        print(f"Attempting to join: {face_target_name} to {pickup_target_name} as {program_name_to_pickup}")
        # Call the plugin command to join the face target to the pickup target
        status_to_pickup = RDK.PluginCommand(
            "CollisionFreePlanner",
            "Join",
            f"{face_target_name}|{pickup_target_name}|{program_name_to_pickup}"
        )
        print(f"Status for '{program_name_to_pickup}': {status_to_pickup}")

        # --- Check and delete existing "From Pickup" program ---
        existing_prog_from_pickup = RDK.Item(program_name_from_pickup, ITEM_TYPE_PROGRAM)
        if existing_prog_from_pickup.Valid():
            print(f"Deleting existing program: {program_name_from_pickup}")
            existing_prog_from_pickup.Delete()

        print(f"Attempting to join: {pickup_target_name} to {face_target_name} as {program_name_from_pickup}")
        # Call the plugin command to join the pickup target to the face target
        status_from_pickup = RDK.PluginCommand(
            "CollisionFreePlanner",
            "Join",
            f"{pickup_target_name}|{face_target_name}|{program_name_from_pickup}"
        )
        print(f"Status for '{program_name_from_pickup}': {status_from_pickup}")


    print("\nPickup link generation process finished.")


# --- Main execution: Run only the new functions ---
if __name__ == '__main__':
    create_face_targets()
    generate_pickup_links()
    create_face_programs()
    addmainprogram()

--- Python program ProgramGenerator ---
from robodk import robolink

# Connect to RoboDK
RDK = robolink.Robolink()

# Get the robot, reference frame, and base point
robot = RDK.Item('UR10e')  # Replace 'Robot' with your robot's name
reference_frame = RDK.Item('CSV Frame')  # Replace 'Reference Frame' with your frame's name
base_point = RDK.Item('Target 33')  # Replace 'Point 1' with your base point's name

# Create a new program
program = RDK.AddProgram('AutoProgram')

# Get all targets under the reference frame
targets = reference_frame.Childs()
target_list = [target for target in targets if target.Type() == robolink.ITEM_TYPE_TARGET]

# Add movements and screwdriver actions to the program
for i, target in enumerate(target_list):
    # Move to the base point first (except for the first target)
    if i > 0:
        program.MoveL(base_point)

    # Move to the target point
    program.MoveL(target)

    # Execute screwdriver actions
    program.RunInstruction('move_shank(20)', robolink.INSTRUCTION_CALL_PROGRAM)  # Tighten screw
    program.RunInstruction('move_shank(0)', robolink.INSTRUCTION_CALL_PROGRAM)  # Release screwdriver

# Save the program
#program.ShowTargets(False)  # Hide targets for clarity
program.Update()
print("Program generated successfully!")

--- Python program ProgramGenerator ---
from robodk import robolink

# Connect to RoboDK
RDK = robolink.Robolink()

# Get the robot, reference frame, and base point
robot = RDK.Item('UR10e')  # Replace 'Robot' with your robot's name
reference_frame = RDK.Item('CSV Frame')  # Replace 'Reference Frame' with your frame's name
base_point = RDK.Item('Target 33')  # Replace 'Point 1' with your base point's name

# Create a new program
program = RDK.AddProgram('AutoProgram')

# Get all targets under the reference frame
targets = reference_frame.Childs()
target_list = [target for target in targets if target.Type() == robolink.ITEM_TYPE_TARGET]

# Add movements and screwdriver actions to the program
for i, target in enumerate(target_list):
    # Move to the base point first (except for the first target)
    if i > 0:
        program.MoveL(base_point)

    # Move to the target point
    program.MoveL(target)

    # Execute screwdriver actions
    program.RunInstruction('move_shank(20)', robolink.INSTRUCTION_CALL_PROGRAM)  # Tighten screw
    program.RunInstruction('move_shank(0)', robolink.INSTRUCTION_CALL_PROGRAM)  # Release screwdriver

# Save the program
#program.ShowTargets(False)  # Hide targets for clarity
program.Update()
print("Program generated successfully!")

--- program pickupm5Totoolswitchm8approach (robot UR10e) ---
  MoveJ (Pt 1 (S1138)) to (-437.91, 304.62, 83.06) mm, rotated rx 148.82 ry 3.26 rz -178.93 deg; joints [-75.565, -105.059, 145.828, -26.927, 13.754, -134.641]
  MoveJ (Pt 2 (S1069)) to (-424.05, 221.6, 32.68) mm, rotated rx 148.94 ry 3.77 rz -174.12 deg; joints [-76.807, -103.326, 153.048, -22.371, 8.218, -148.169]
  MoveJ (Pt 3 (S995)) to (-436.51, 254.57, 169.63) mm, rotated rx 148.94 ry 3.77 rz -174.12 deg; joints [-75.55, -113.946, 140.961, -3.178, 9.351, -144.613]
  MoveJ (Pt 4 (S1013)) to (-349.4, 349.66, 227.68) mm, rotated rx 175.61 ry -30.98 rz 98.15 deg; joints [-40.94, -114.594, 151.115, -74.991, 124.156, -118.436]
  MoveJ (Pt 5 (S876)) to (-566.01, -9.66, 385.13) mm, rotated rx 90 ry -10 rz -90 deg; joints [-56.219, -97.868, 132.397, -22.553, -56.798, -186.625]
  MoveJ (Pt 6 (S768)) to (-566.01, -53.07, 388.93) mm, rotated rx 90 ry 0 rz -90 deg; joints [-52.421, -105.764, 133.113, -27.35, -52.42, -179.999]
  MoveJ (Pt 7 (S516)) to (-566.01, -172.58, 395.39) mm, rotated rx 90 ry 0 rz -90 deg; joints [-37.286, -110.687, 135.476, -24.792, -37.284, -179.998]
  MoveJ (Pt 8 (S386)) to (-566.01, -242.72, 394.37) mm, rotated rx 90 ry 0 rz -90 deg; joints [-25.901, -110.898, 135.712, -24.817, -25.9, -179.997]
  MoveJ (Pt 9 (S229)) to (-566.01, -361.29, 394.37) mm, rotated rx 90 ry 0 rz -90 deg; joints [-5.068, -107.128, 133.402, -26.287, -5.067, -179.986]
  MoveJ (Pt 10 (S154)) to (-816.01, -361.29, 394.37) mm, rotated rx 90 ry 0 rz -90 deg; joints [-2.904, -81.882, 110.532, -28.675, -2.903, -179.976]
  MoveJ (Pt 11 (S109)) to (-816.02, -422.58, 395.39) mm, rotated rx 90 ry 0 rz -90 deg; joints [2.982, -80.355, 108.601, -28.223, 2.983, -180.023]
  MoveJ (Pt 12 (S93)) to (-624.17, -467.56, 176.05) mm, rotated rx -179.87 ry 0.01 rz -89.96 deg; joints [6.858, -76.682, 103.853, 332.885, 6.813, -89.924]
  MoveJ (Pt 13 (S142)) to (-623.94, -467.54, 76.05) mm, rotated rx -179.87 ry 0.01 rz -89.96 deg; joints [6.859, -71.505, 108.744, 322.817, 6.815, -89.924]

--- program Program_Main_Combined_met (robot UR10e) ---
  Set Tool: schroevendraaier all in met nieuw kopstuk en tool
  Set Ref.: CSV Frame
  Call pickupm8Totoolswitchm8approach
  Call toolswitchm8approachTopickupm8
  Call Program_Main_m8
  Call pickupm8Totoolswitchm8approach
  Call toolswitchm8approachTopickupm8

--- program Program_Main_Combined_met (robot UR10e) ---
  Set Tool: schroevendraaier all in met nieuw kopstuk en tool
  Set Ref.: CSV Frame
  Call pickupm8Totoolswitchm8approach
  MoveL (toolswitch_m8)
  Call screw_out(0)
  MoveL (toolswitch_m8_approach)
  Call toolswitchm8approachTopickupm8
  Call Program_Main_m8
  Call pickupm8Totoolswitchm8approach
  MoveL (toolswitch_m8)
  Call screw_in(10)
  MoveL (toolswitch_m8_approach)
  Call toolswitchm8approachTopickupm8

--- program Program_Main_Combined_met (robot UR10e) ---
  Set Tool: schroevendraaier all in met nieuw kopstuk en tool
  Set Ref.: CSV Frame

--- program Prog43 (robot UR10e) ---
  Set Ref.: CSV Frame
  Set Tool: schroevendraaier all in met nieuw kopstuk en tool
  MoveL (toolswitch_m8_approach)
  MoveL (toolswitch_m8)
  Call screw_out(0)
  MoveL (toolswitch_m8_approach)
  MoveL (toolswitch_m8_approach)
  MoveL (toolswitch_m8)
  Call screw_in(10)
  MoveL (toolswitch_m8_approach)

--- program pickupm8Totoolswitchm8 (robot UR10e) ---
  MoveJ (Pt 1 (S1265)) to (-361.97, 306.04, 87.38) mm, rotated rx 148.82 ry 3.26 rz -178.93 deg; joints [-96.274, -127.938, 155.828, 308.074, -8.028, -97.355]
  MoveJ (Pt 2 (S1276)) to (-291.81, 189.68, 43.36) mm, rotated rx 173.25 ry 30.68 rz -107.38 deg; joints [-75.824, -114.001, 145.678, 293.478, -63.249, -79.354]
  MoveJ (Pt 3 (S1105)) to (-362.69, 295.7, 104.49) mm, rotated rx 173.25 ry 30.68 rz -107.38 deg; joints [-70.201, -101.671, 131.181, 293.82, -58.685, -75.597]
  MoveJ (Pt 4 (S1048)) to (-433.56, 401.71, 165.63) mm, rotated rx 173.25 ry 30.68 rz -107.38 deg; joints [-67.129, -91.484, 115.69, 297.937, -56.239, -73.391]
  MoveJ (Pt 5 (S1116)) to (-437.47, 349.85, 251.04) mm, rotated rx 173.25 ry 30.68 rz -107.38 deg; joints [-64.592, -98.205, 112.824, 306.43, -54.251, -71.473]
  MoveJ (Pt 6 (S1022)) to (-463.16, 267.77, 200.01) mm, rotated rx 173.25 ry 30.68 rz -107.38 deg; joints [-57.766, -100.913, 120.893, 297.542, -49.071, -65.796]
  MoveJ (Pt 7 (S999)) to (-488.86, 185.69, 148.99) mm, rotated rx 173.25 ry 30.68 rz -107.38 deg; joints [-49.635, -101.874, 128.097, 285.751, -43.336, -57.797]
  MoveJ (Pt 8 (S918)) to (-484.94, 237.56, 63.59) mm, rotated rx 173.25 ry 30.68 rz -107.38 deg; joints [-53.767, -93.623, 130.789, 277.833, -46.181, -62.054]
  MoveJ (Pt 9 (S905)) to (-484.22, 247.88, 46.49) mm, rotated rx 173.24 ry 30.67 rz -107.38 deg; joints [-54.525, -91.744, 131.117, 276.144, -46.717, -62.802]
  MoveJ (Pt 10 (S31)) to (-569.54, 226.04, 79.52) mm, rotated rx -176.96 ry 3.26 rz -178.93 deg; joints [-56.803, -92.592, 131.94, -33.233, 32.278, -92.138]
  MoveJ (Pt 11 (S27)) to (-580.12, 225.84, 78.92) mm, rotated rx -176.96 ry 3.26 rz -178.93 deg; joints [-55.548, -91.667, 131.136, -33.557, 33.527, -91.896]
  MoveJ (Pt 12 (S28)) to (-581.67, 325.69, 73.63) mm, rotated rx -176.96 ry 3.26 rz -178.93 deg; joints [-62.052, -84.921, 124.838, -32.736, 27.065, -93.365]

--- program toolswitchm8Topickupm8 (robot UR10e) ---
  MoveJ (Pt 1 (S28)) to (-581.67, 325.69, 73.63) mm, rotated rx -176.96 ry 3.26 rz -178.93 deg; joints [-62.052, -84.921, 124.838, -32.736, 27.065, -93.365]
  MoveJ (Pt 2 (S27)) to (-580.12, 225.84, 78.92) mm, rotated rx -176.96 ry 3.26 rz -178.93 deg; joints [-55.548, -91.667, 131.136, -33.557, 33.527, -91.896]
  MoveJ (Pt 3 (S31)) to (-569.54, 226.04, 79.52) mm, rotated rx -176.96 ry 3.26 rz -178.93 deg; joints [-56.803, -92.592, 131.94, -33.233, 32.278, -92.138]
  MoveJ (Pt 4 (S905)) to (-484.22, 247.88, 46.49) mm, rotated rx 173.24 ry 30.67 rz -107.38 deg; joints [-54.525, -91.744, 131.117, 276.144, -46.717, -62.802]
  MoveJ (Pt 5 (S975)) to (-488.13, 196.03, 131.91) mm, rotated rx 173.24 ry 30.67 rz -107.38 deg; joints [-50.502, -100.38, 128.761, 284.277, -43.917, -58.739]
  MoveJ (Pt 6 (S999)) to (-488.86, 185.69, 148.99) mm, rotated rx 173.25 ry 30.68 rz -107.38 deg; joints [-49.635, -101.874, 128.097, 285.751, -43.336, -57.797]
  MoveJ (Pt 7 (S1022)) to (-463.16, 267.77, 200.01) mm, rotated rx 173.25 ry 30.68 rz -107.38 deg; joints [-57.766, -100.913, 120.893, 297.542, -49.071, -65.796]
  MoveJ (Pt 8 (S1116)) to (-437.47, 349.85, 251.04) mm, rotated rx 173.25 ry 30.68 rz -107.38 deg; joints [-64.592, -98.205, 112.824, 306.43, -54.251, -71.473]
  MoveJ (Pt 9 (S1048)) to (-433.56, 401.71, 165.63) mm, rotated rx 173.25 ry 30.68 rz -107.38 deg; joints [-67.129, -91.484, 115.69, 297.937, -56.239, -73.391]
  MoveJ (Pt 10 (S1105)) to (-362.69, 295.7, 104.49) mm, rotated rx 173.25 ry 30.68 rz -107.38 deg; joints [-70.201, -101.671, 131.181, 293.82, -58.685, -75.597]
  MoveJ (Pt 11 (S1276)) to (-291.81, 189.68, 43.36) mm, rotated rx 173.25 ry 30.68 rz -107.38 deg; joints [-75.824, -114.001, 145.678, 293.478, -63.249, -79.354]
  MoveJ (Pt 12 (S1265)) to (-361.97, 306.04, 87.38) mm, rotated rx 148.82 ry 3.26 rz -178.93 deg; joints [-96.274, -127.938, 155.828, 308.074, -8.028, -97.355]

--- program pickupm5Totoolswitchm5 (robot UR10e) ---
  MoveJ (Pt 1 (S136)) to (-437.91, 304.62, 83.06) mm, rotated rx 148.82 ry 3.26 rz -178.93 deg; joints [-75.565, -105.059, 145.828, -26.927, 13.754, -134.641]
  MoveJ (Pt 2 (S153)) to (-441.81, 252.77, 168.47) mm, rotated rx 148.82 ry 3.26 rz -178.93 deg; joints [-70.855, -118.095, 142.384, -13.886, 18.361, -131.066]
  MoveJ (Pt 3 (S131)) to (-437.28, 167.28, 116.78) mm, rotated rx 148.82 ry 3.26 rz -178.93 deg; joints [-61.41, -123.306, 150.061, -19.726, 27.701, -127.411]
  MoveJ (Pt 4 (S89)) to (-536.97, 244.32, 163.05) mm, rotated rx 148.94 ry 3.76 rz -174.12 deg; joints [-54.5, -105.959, 136.001, -22.458, 29.834, -127.646]
  MoveJ (Pt 5 (S83)) to (-546.17, 336.39, 214.47) mm, rotated rx 148.82 ry 3.26 rz -178.93 deg; joints [-59.094, -102.782, 128.155, -18.841, 30.001, -126.844]
  MoveJ (Pt 6 (S41)) to (-575.31, 231.23, 179.22) mm, rotated rx -176.96 ry 3.26 rz -178.93 deg; joints [-56.524, -98.258, 124.969, -20.643, 32.555, -92.082]
  MoveJ (Pt 7 (S35)) to (-585.89, 231.03, 178.62) mm, rotated rx -176.96 ry 3.26 rz -178.93 deg; joints [-55.298, -97.308, 124.236, -21.056, 33.775, -91.849]
  MoveJ (Pt 8 (S30)) to (-687.27, 329.02, 167.64) mm, rotated rx -176.96 ry 3.26 rz -178.93 deg; joints [-52.489, -83.001, 111.208, -22.729, 36.57, -91.367]
  MoveJ (Pt 9 (S4)) to (-681.49, 323.83, 67.94) mm, rotated rx -176.96 ry 3.26 rz -178.93 deg; joints [-52.635, -78.013, 117.195, -33.685, 36.425, -91.391]
  MoveJ (Pt 10 (S3)) to (-670.91, 324.03, 68.54) mm, rotated rx -176.96 ry 3.26 rz -178.93 deg; joints [-53.522, -78.759, 118.074, -33.7, 35.542, -91.537]

--- program toolswitchm5Topickupm5 (robot UR10e) ---
  MoveJ (Pt 1 (S3)) to (-670.91, 324.03, 68.54) mm, rotated rx -176.96 ry 3.26 rz -178.93 deg; joints [-53.522, -78.759, 118.074, -33.7, 35.542, -91.537]
  MoveJ (Pt 2 (S4)) to (-681.49, 323.83, 67.94) mm, rotated rx -176.96 ry 3.26 rz -178.93 deg; joints [-52.635, -78.013, 117.195, -33.685, 36.425, -91.391]
  MoveJ (Pt 3 (S30)) to (-687.27, 329.02, 167.64) mm, rotated rx -176.96 ry 3.26 rz -178.93 deg; joints [-52.489, -83.001, 111.208, -22.729, 36.57, -91.367]
  MoveJ (Pt 4 (S35)) to (-585.89, 231.03, 178.62) mm, rotated rx -176.96 ry 3.26 rz -178.93 deg; joints [-55.298, -97.308, 124.236, -21.056, 33.775, -91.849]
  MoveJ (Pt 5 (S41)) to (-575.31, 231.23, 179.22) mm, rotated rx -176.96 ry 3.26 rz -178.93 deg; joints [-56.524, -98.258, 124.969, -20.643, 32.555, -92.082]
  MoveJ (Pt 6 (S83)) to (-546.17, 336.39, 214.47) mm, rotated rx 148.82 ry 3.26 rz -178.93 deg; joints [-59.094, -102.782, 128.155, -18.841, 30.001, -126.844]
  MoveJ (Pt 7 (S89)) to (-536.97, 244.32, 163.05) mm, rotated rx 148.94 ry 3.76 rz -174.12 deg; joints [-54.5, -105.959, 136.001, -22.458, 29.834, -127.646]
  MoveJ (Pt 8 (S131)) to (-437.28, 167.28, 116.78) mm, rotated rx 148.82 ry 3.26 rz -178.93 deg; joints [-61.41, -123.306, 150.061, -19.726, 27.701, -127.411]
  MoveJ (Pt 9 (S153)) to (-441.81, 252.77, 168.47) mm, rotated rx 148.82 ry 3.26 rz -178.93 deg; joints [-70.855, -118.095, 142.384, -13.886, 18.361, -131.066]
  MoveJ (Pt 10 (S136)) to (-437.91, 304.62, 83.06) mm, rotated rx 148.82 ry 3.26 rz -178.93 deg; joints [-75.565, -105.059, 145.828, -26.927, 13.754, -134.641]

--- program FaceTarget0ToPickupm8 (robot UR10e) ---
  MoveJ (Pt 1 (S1239)) to (-816.01, -159.97, 145.4) mm, rotated rx 90 ry 0 rz -90 deg; joints [-22.389, -65.52, 121.579, 303.939, -22.388, -179.997]
  MoveJ (Pt 2 (S1249)) to (-816.01, -111.28, 144.37) mm, rotated rx 90 ry 0 rz -90 deg; joints [-26.792, -65.006, 120.835, 304.168, -26.791, -179.998]
  MoveJ (Pt 3 (S1043)) to (-433.56, 401.71, 165.63) mm, rotated rx 173.25 ry 30.68 rz -107.38 deg; joints [-67.129, -91.484, 115.69, 297.937, -56.239, -73.391]
  MoveJ (Pt 4 (S1095)) to (-362.69, 295.7, 104.49) mm, rotated rx 173.25 ry 30.68 rz -107.38 deg; joints [-70.201, -101.671, 131.181, 293.82, -58.685, -75.597]
  MoveJ (Pt 5 (S1259)) to (-291.81, 189.68, 43.36) mm, rotated rx 173.25 ry 30.68 rz -107.38 deg; joints [-75.824, -114.001, 145.678, 293.478, -63.249, -79.354]
  MoveJ (Pt 6 (S1245)) to (-361.97, 306.04, 87.38) mm, rotated rx 148.82 ry 3.26 rz -178.93 deg; joints [-96.274, -127.938, 155.828, 308.074, -8.028, -97.355]

--- program Pickupm8ToFaceTarget0 (robot UR10e) ---
  MoveJ (Pt 1 (S1245)) to (-361.97, 306.04, 87.38) mm, rotated rx 148.82 ry 3.26 rz -178.93 deg; joints [-96.274, -127.938, 155.828, 308.074, -8.028, -97.355]
  MoveJ (Pt 2 (S1259)) to (-291.81, 189.68, 43.36) mm, rotated rx 173.25 ry 30.68 rz -107.38 deg; joints [-75.824, -114.001, 145.678, 293.478, -63.249, -79.354]
  MoveJ (Pt 3 (S1095)) to (-362.69, 295.7, 104.49) mm, rotated rx 173.25 ry 30.68 rz -107.38 deg; joints [-70.201, -101.671, 131.181, 293.82, -58.685, -75.597]
  MoveJ (Pt 4 (S1043)) to (-433.56, 401.71, 165.63) mm, rotated rx 173.25 ry 30.68 rz -107.38 deg; joints [-67.129, -91.484, 115.69, 297.937, -56.239, -73.391]
  MoveJ (Pt 5 (S1249)) to (-816.01, -111.28, 144.37) mm, rotated rx 90 ry 0 rz -90 deg; joints [-26.792, -65.006, 120.835, 304.168, -26.791, -179.998]
  MoveJ (Pt 6 (S1239)) to (-816.01, -159.97, 145.4) mm, rotated rx 90 ry 0 rz -90 deg; joints [-22.389, -65.52, 121.579, 303.939, -22.388, -179.997]

--- program FaceTarget1ToPickupm8 (robot UR10e) ---
  MoveJ (Pt 1 (S1390)) to (-910.43, -13.22, 388.49) mm, rotated rx 135 ry 0 rz -90 deg; joints [-28.011, -71.089, 80.867, 350.219, -28.01, -134.998]
  MoveJ (Pt 2 (S1381)) to (-910.43, -56.47, 388.49) mm, rotated rx 135 ry 0 rz -90 deg; joints [-25.08, -72.06, 82.172, 349.885, -25.079, -134.997]
  MoveJ (Pt 3 (S1127)) to (-539.86, 560.74, 257.33) mm, rotated rx 173.25 ry 30.68 rz -107.38 deg; joints [-64.444, -76.48, 89.354, 308.108, -54.136, -71.358]
  MoveJ (Pt 4 (S1113)) to (-437.47, 349.85, 251.04) mm, rotated rx 173.25 ry 30.68 rz -107.38 deg; joints [-64.592, -98.205, 112.824, 306.43, -54.251, -71.473]
  MoveJ (Pt 5 (S1043)) to (-433.56, 401.71, 165.63) mm, rotated rx 173.25 ry 30.68 rz -107.38 deg; joints [-67.129, -91.484, 115.69, 297.937, -56.239, -73.391]
  MoveJ (Pt 6 (S1095)) to (-362.69, 295.7, 104.49) mm, rotated rx 173.25 ry 30.68 rz -107.38 deg; joints [-70.201, -101.671, 131.181, 293.82, -58.685, -75.597]
  MoveJ (Pt 7 (S1259)) to (-291.81, 189.68, 43.36) mm, rotated rx 173.25 ry 30.68 rz -107.38 deg; joints [-75.824, -114.001, 145.678, 293.478, -63.249, -79.354]
  MoveJ (Pt 8 (S1245)) to (-361.97, 306.04, 87.38) mm, rotated rx 148.82 ry 3.26 rz -178.93 deg; joints [-96.274, -127.938, 155.828, 308.074, -8.028, -97.355]

--- program Pickupm8ToFaceTarget1 (robot UR10e) ---
  MoveJ (Pt 1 (S1245)) to (-361.97, 306.04, 87.38) mm, rotated rx 148.82 ry 3.26 rz -178.93 deg; joints [-96.274, -127.938, 155.828, 308.074, -8.028, -97.355]
  MoveJ (Pt 2 (S1259)) to (-291.81, 189.68, 43.36) mm, rotated rx 173.25 ry 30.68 rz -107.38 deg; joints [-75.824, -114.001, 145.678, 293.478, -63.249, -79.354]
  MoveJ (Pt 3 (S1095)) to (-362.69, 295.7, 104.49) mm, rotated rx 173.25 ry 30.68 rz -107.38 deg; joints [-70.201, -101.671, 131.181, 293.82, -58.685, -75.597]
  MoveJ (Pt 4 (S1043)) to (-433.56, 401.71, 165.63) mm, rotated rx 173.25 ry 30.68 rz -107.38 deg; joints [-67.129, -91.484, 115.69, 297.937, -56.239, -73.391]
  MoveJ (Pt 5 (S1113)) to (-437.47, 349.85, 251.04) mm, rotated rx 173.25 ry 30.68 rz -107.38 deg; joints [-64.592, -98.205, 112.824, 306.43, -54.251, -71.473]
  MoveJ (Pt 6 (S1127)) to (-539.86, 560.74, 257.33) mm, rotated rx 173.25 ry 30.68 rz -107.38 deg; joints [-64.444, -76.48, 89.354, 308.108, -54.136, -71.358]
  MoveJ (Pt 7 (S1381)) to (-910.43, -56.47, 388.49) mm, rotated rx 135 ry 0 rz -90 deg; joints [-25.08, -72.06, 82.172, 349.885, -25.079, -134.997]
  MoveJ (Pt 8 (S1390)) to (-910.43, -13.22, 388.49) mm, rotated rx 135 ry 0 rz -90 deg; joints [-28.011, -71.089, 80.867, 350.219, -28.01, -134.998]

--- program FaceTarget2ToPickupm8 (robot UR10e) ---
  MoveJ (Pt 1 (S1558)) to (-1103.52, -62.25, 481.99) mm, rotated rx 180 ry 0 rz 173.43 deg; joints [-5.588, -58.826, 71.227, 167.599, -90.985, -270.001]
  MoveJ (Pt 2 (S1535)) to (-1100.79, -83.02, 481.99) mm, rotated rx 180 ry 0 rz 180 deg; joints [-5.882, -59.281, 71.94, 167.342, -84.119, -270.001]
  MoveJ (Pt 3 (S1520)) to (-1086.49, -83.02, 481.99) mm, rotated rx 180 ry 0 rz 180 deg; joints [-5.98, -60.665, 74.085, 166.58, -84.021, -270.001]
  MoveJ (Pt 4 (S1500)) to (-1087.69, 17.1, 481.99) mm, rotated rx -180 ry 0 rz 180 deg; joints [-12.597, -60.926, 74.486, 166.439, -77.405, -270]
  MoveJ (Pt 5 (S1195)) to (-837.69, 167.09, 482) mm, rotated rx -180 ry 0 rz 180 deg; joints [-30.714, -82.014, 103.063, 158.95, -59.288, -270]
  MoveJ (Pt 6 (S1194)) to (-836.49, 166.97, 482) mm, rotated rx 180 ry 0 rz 180 deg; joints [-30.761, -82.125, 103.192, 158.933, -59.241, -270.001]
  MoveJ (Pt 7 (S346)) to (-816.01, -53.06, 38.93) mm, rotated rx 90 ry 0 rz -90 deg; joints [-31.756, -54.307, 119.94, -65.636, -31.755, -179.998]
  MoveJ (Pt 8 (S398)) to (-716.01, -140.46, 38.93) mm, rotated rx 90 ry 0 rz -90 deg; joints [-29.092, -59.226, 133.248, -74.024, -29.09, -179.998]
  MoveJ (Pt 9 (S392)) to (-716.01, -142.71, 44.37) mm, rotated rx 90 ry 0 rz -90 deg; joints [-28.852, -59.911, 133.311, -73.402, -28.85, -179.998]
  MoveJ (Pt 10 (S277)) to (-716.01, -140.46, 138.93) mm, rotated rx 90 ry 0 rz -90 deg; joints [-29.091, -71.077, 132.642, -61.568, -29.09, -179.998]
  MoveJ (Pt 11 (S227)) to (-716.01, -140.46, 238.93) mm, rotated rx 90 ry 0 rz -90 deg; joints [-29.091, -81.291, 129.875, -48.586, -29.09, -179.998]
  MoveJ (Pt 12 (S1231)) to (-239.71, 364.19, 128.27) mm, rotated rx 173.24 ry 30.67 rz -107.38 deg; joints [-87.692, -103.504, 129.241, 302.057, -73.157, -86.413]
  MoveJ (Pt 13 (S1255)) to (-265.4, 282.1, 77.27) mm, rotated rx 173.24 ry 30.67 rz -107.38 deg; joints [-83.109, -108.057, 138.191, 296.821, -69.296, -83.804]
  MoveJ (Pt 14 (S1222)) to (-291.09, 200.02, 26.26) mm, rotated rx 173.24 ry 30.67 rz -107.38 deg; joints [-76.418, -111.273, 146.328, 290.278, -63.737, -79.741]
  MoveJ (Pt 15 (S1245)) to (-361.97, 306.04, 87.38) mm, rotated rx 148.82 ry 3.26 rz -178.93 deg; joints [-96.274, -127.938, 155.828, 308.074, -8.028, -97.355]

--- program Pickupm8ToFaceTarget2 (robot UR10e) ---
  MoveJ (Pt 1 (S1245)) to (-361.97, 306.04, 87.38) mm, rotated rx 148.82 ry 3.26 rz -178.93 deg; joints [-96.274, -127.938, 155.828, 308.074, -8.028, -97.355]
  MoveJ (Pt 2 (S1222)) to (-291.09, 200.02, 26.26) mm, rotated rx 173.24 ry 30.67 rz -107.38 deg; joints [-76.418, -111.273, 146.328, 290.278, -63.737, -79.741]
  MoveJ (Pt 3 (S1255)) to (-265.4, 282.1, 77.27) mm, rotated rx 173.24 ry 30.67 rz -107.38 deg; joints [-83.109, -108.057, 138.191, 296.821, -69.296, -83.804]
  MoveJ (Pt 4 (S1231)) to (-239.71, 364.19, 128.27) mm, rotated rx 173.24 ry 30.67 rz -107.38 deg; joints [-87.692, -103.504, 129.241, 302.057, -73.157, -86.413]
  MoveJ (Pt 5 (S227)) to (-716.01, -140.46, 238.93) mm, rotated rx 90 ry 0 rz -90 deg; joints [-29.091, -81.291, 129.875, -48.586, -29.09, -179.998]
  MoveJ (Pt 6 (S277)) to (-716.01, -140.46, 138.93) mm, rotated rx 90 ry 0 rz -90 deg; joints [-29.091, -71.077, 132.642, -61.568, -29.09, -179.998]
  MoveJ (Pt 7 (S392)) to (-716.01, -142.71, 44.37) mm, rotated rx 90 ry 0 rz -90 deg; joints [-28.852, -59.911, 133.311, -73.402, -28.85, -179.998]
  MoveJ (Pt 8 (S398)) to (-716.01, -140.46, 38.93) mm, rotated rx 90 ry 0 rz -90 deg; joints [-29.092, -59.226, 133.248, -74.024, -29.09, -179.998]
  MoveJ (Pt 9 (S346)) to (-816.01, -53.06, 38.93) mm, rotated rx 90 ry 0 rz -90 deg; joints [-31.756, -54.307, 119.94, -65.636, -31.755, -179.998]
  MoveJ (Pt 10 (S1194)) to (-836.49, 166.97, 482) mm, rotated rx 180 ry 0 rz 180 deg; joints [-30.761, -82.125, 103.192, 158.933, -59.241, -270.001]
  MoveJ (Pt 11 (S1195)) to (-837.69, 167.09, 482) mm, rotated rx -180 ry 0 rz 180 deg; joints [-30.714, -82.014, 103.063, 158.95, -59.288, -270]
  MoveJ (Pt 12 (S1522)) to (-1087.69, -82.9, 481.99) mm, rotated rx -180 ry 0 rz 180 deg; joints [-5.98, -60.551, 73.909, 166.641, -84.022, -270]
  MoveJ (Pt 13 (S1535)) to (-1100.79, -83.02, 481.99) mm, rotated rx 180 ry 0 rz 180 deg; joints [-5.882, -59.281, 71.94, 167.342, -84.119, -270.001]
  MoveJ (Pt 14 (S1558)) to (-1103.52, -62.25, 481.99) mm, rotated rx 180 ry 0 rz 173.43 deg; joints [-5.588, -58.826, 71.227, 167.599, -90.985, -270.001]

--- program Program_Face_0_m8 (robot UR10e) ---
  Call screw_in(0)
  Call Pickupm8ToFaceTarget0
  MoveL (Face_Target_0)
  MoveL (H-8.3_15.0-1)
  Call screw_in(20)
  Call screw_out(0)
  MoveL (Face_Target_0)
  Call FaceTarget0ToPickupm8
  Call screw_in(0)
  Call Pickupm8ToFaceTarget0
  MoveL (Face_Target_0)
  MoveL (H-8.3_15.0-2)
  Call screw_in(20)
  Call screw_out(0)
  MoveL (Face_Target_0)
  Call FaceTarget0ToPickupm8
  Call screw_in(0)

--- program Program_Face_1_m8 (robot UR10e) ---
  Call Pickupm8ToFaceTarget1
  MoveL (Face_Target_1)
  MoveL (H-8.3_15.0-9)
  Call screw_in(20)
  Call screw_out(0)
  MoveL (Face_Target_1)
  Call FaceTarget1ToPickupm8
  Call screw_in(0)
  Call Pickupm8ToFaceTarget1
  MoveL (Face_Target_1)
  MoveL (H-8.3_15.0-11)
  Call screw_in(20)
  Call screw_out(0)
  MoveL (Face_Target_1)
  Call FaceTarget1ToPickupm8
  Call screw_in(0)

--- program Program_Face_2_m8 (robot UR10e) ---
  Call Pickupm8ToFaceTarget2
  MoveL (Face_Target_2)
  MoveL (H-8.3_15.0-16)
  Call screw_in(20)
  Call screw_out(0)
  MoveL (Face_Target_2)
  Call FaceTarget2ToPickupm8
  Call screw_in(0)
  Call Pickupm8ToFaceTarget2
  MoveL (Face_Target_2)
  MoveL (H-8.3_15.0-17)
  Call screw_in(20)
  Call screw_out(0)
  MoveL (Face_Target_2)
  Call FaceTarget2ToPickupm8

--- program FaceTarget0ToPickupm5 (robot UR10e) ---
  MoveJ (Pt 1 (S1239)) to (-816.01, -159.97, 145.4) mm, rotated rx 90 ry 0 rz -90 deg; joints [-22.389, -65.52, 121.579, 303.939, -22.388, -179.997]
  MoveJ (Pt 2 (S1233)) to (-816.01, -172.57, 145.39) mm, rotated rx 90 ry 0 rz -90 deg; joints [-21.218, -65.589, 121.702, 303.884, -21.217, -179.997]
  MoveJ (Pt 3 (S1232)) to (-816.01, -259.97, 145.39) mm, rotated rx 90 ry 0 rz -90 deg; joints [-12.834, -65.597, 121.717, 303.875, -12.833, -179.995]
  MoveJ (Pt 4 (S1217)) to (-816.01, -259.97, 45.39) mm, rotated rx 90 ry 0 rz -90 deg; joints [-12.835, -55.909, 122.365, 293.538, -12.833, -179.995]
  MoveJ (Pt 5 (S1209)) to (-716.01, -259.97, 45.39) mm, rotated rx 90 ry 0 rz -90 deg; joints [-15.54, -60.182, 133.733, 286.444, -15.539, -179.996]
  MoveJ (Pt 6 (S1223)) to (-716.01, -259.97, 145.39) mm, rotated rx 90 ry 0 rz -90 deg; joints [-15.54, -72.064, 132.978, 299.082, -15.539, -179.996]
  MoveJ (Pt 7 (S1220)) to (-716.01, -159.97, 145.4) mm, rotated rx 90 ry 0 rz -90 deg; joints [-26.989, -71.969, 132.818, 299.149, -26.987, -179.998]
  MoveJ (Pt 8 (S1273)) to (-716.01, -98.69, 181.83) mm, rotated rx 90 ry 0 rz -90 deg; joints [-33.401, -75.109, 130.821, 304.286, -33.399, -179.998]
  MoveJ (Pt 9 (S1100)) to (-556.88, -13.22, 34.94) mm, rotated rx 135 ry 0 rz -90 deg; joints [-49.771, -80.79, 137.167, 303.621, -49.77, -134.999]
  MoveJ (Pt 10 (S994)) to (-457.25, 218.7, 30) mm, rotated rx 148.82 ry 3.26 rz -178.93 deg; joints [-63.329, -105.109, 152.954, 319.665, 25.798, -127.95]
  MoveJ (Pt 11 (S195)) to (-424.05, 221.6, 32.68) mm, rotated rx 148.94 ry 3.77 rz -174.12 deg; joints [-76.807, -103.326, 153.048, -22.371, 8.218, -148.169]
  MoveJ (Pt 12 (S136)) to (-437.91, 304.62, 83.06) mm, rotated rx 148.82 ry 3.26 rz -178.93 deg; joints [-75.565, -105.059, 145.828, -26.927, 13.754, -134.641]

--- program Pickupm5ToFaceTarget0 (robot UR10e) ---
  MoveJ (Pt 1 (S136)) to (-437.91, 304.62, 83.06) mm, rotated rx 148.82 ry 3.26 rz -178.93 deg; joints [-75.565, -105.059, 145.828, -26.927, 13.754, -134.641]
  MoveJ (Pt 2 (S195)) to (-424.05, 221.6, 32.68) mm, rotated rx 148.94 ry 3.77 rz -174.12 deg; joints [-76.807, -103.326, 153.048, -22.371, 8.218, -148.169]
  MoveJ (Pt 3 (S994)) to (-457.25, 218.7, 30) mm, rotated rx 148.82 ry 3.26 rz -178.93 deg; joints [-63.329, -105.109, 152.954, 319.665, 25.798, -127.95]
  MoveJ (Pt 4 (S1100)) to (-556.88, -13.22, 34.94) mm, rotated rx 135 ry 0 rz -90 deg; joints [-49.771, -80.79, 137.167, 303.621, -49.77, -134.999]
  MoveJ (Pt 5 (S1273)) to (-716.01, -98.69, 181.83) mm, rotated rx 90 ry 0 rz -90 deg; joints [-33.401, -75.109, 130.821, 304.286, -33.399, -179.998]
  MoveJ (Pt 6 (S1220)) to (-716.01, -159.97, 145.4) mm, rotated rx 90 ry 0 rz -90 deg; joints [-26.989, -71.969, 132.818, 299.149, -26.987, -179.998]
  MoveJ (Pt 7 (S1223)) to (-716.01, -259.97, 145.39) mm, rotated rx 90 ry 0 rz -90 deg; joints [-15.54, -72.064, 132.978, 299.082, -15.539, -179.996]
  MoveJ (Pt 8 (S1209)) to (-716.01, -259.97, 45.39) mm, rotated rx 90 ry 0 rz -90 deg; joints [-15.54, -60.182, 133.733, 286.444, -15.539, -179.996]
  MoveJ (Pt 9 (S1217)) to (-816.01, -259.97, 45.39) mm, rotated rx 90 ry 0 rz -90 deg; joints [-12.835, -55.909, 122.365, 293.538, -12.833, -179.995]
  MoveJ (Pt 10 (S1232)) to (-816.01, -259.97, 145.39) mm, rotated rx 90 ry 0 rz -90 deg; joints [-12.834, -65.597, 121.717, 303.875, -12.833, -179.995]
  MoveJ (Pt 11 (S1233)) to (-816.01, -172.57, 145.39) mm, rotated rx 90 ry 0 rz -90 deg; joints [-21.218, -65.589, 121.702, 303.884, -21.217, -179.997]
  MoveJ (Pt 12 (S1239)) to (-816.01, -159.97, 145.4) mm, rotated rx 90 ry 0 rz -90 deg; joints [-22.389, -65.52, 121.579, 303.939, -22.388, -179.997]

--- program FaceTarget1ToPickupm5 (robot UR10e) ---
  MoveJ (Pt 1 (S1390)) to (-910.43, -13.22, 388.49) mm, rotated rx 135 ry 0 rz -90 deg; joints [-28.011, -71.089, 80.867, 350.219, -28.01, -134.998]
  MoveJ (Pt 2 (S1377)) to (-910.43, -113.22, 388.49) mm, rotated rx 135 ry 0 rz -90 deg; joints [-21.07, -72.993, 83.411, 349.579, -21.069, -134.997]
  MoveJ (Pt 3 (S1426)) to (-839.72, -113.23, 459.2) mm, rotated rx 135 ry 0 rz -90 deg; joints [-23.236, -80.609, 85.748, 354.857, -23.235, -134.997]
  MoveJ (Pt 4 (S1557)) to (-816.01, -159.98, 645.4) mm, rotated rx 90 ry 0 rz -90 deg; joints [-22.388, -89.789, 92.704, 357.083, -22.387, -179.997]
  MoveJ (Pt 5 (S1415)) to (-816.01, -159.98, 395.4) mm, rotated rx 90 ry 0 rz -90 deg; joints [-22.388, -83.255, 112.006, 331.246, -22.387, -179.997]
  MoveJ (Pt 6 (S1320)) to (-716.01, -159.98, 245.4) mm, rotated rx 90 ry 0 rz -90 deg; joints [-26.988, -82.105, 129.904, 312.198, -26.987, -179.998]
  MoveJ (Pt 7 (S1304)) to (-716.01, -59.98, 245.4) mm, rotated rx 90 ry 0 rz -90 deg; joints [-37.136, -80.295, 127.654, 312.639, -37.135, -179.998]
  MoveJ (Pt 8 (S1273)) to (-716.01, -98.69, 181.83) mm, rotated rx 90 ry 0 rz -90 deg; joints [-33.401, -75.109, 130.821, 304.286, -33.399, -179.998]
  MoveJ (Pt 9 (S1100)) to (-556.88, -13.22, 34.94) mm, rotated rx 135 ry 0 rz -90 deg; joints [-49.771, -80.79, 137.167, 303.621, -49.77, -134.999]
  MoveJ (Pt 10 (S994)) to (-457.25, 218.7, 30) mm, rotated rx 148.82 ry 3.26 rz -178.93 deg; joints [-63.329, -105.109, 152.954, 319.665, 25.798, -127.95]
  MoveJ (Pt 11 (S195)) to (-424.05, 221.6, 32.68) mm, rotated rx 148.94 ry 3.77 rz -174.12 deg; joints [-76.807, -103.326, 153.048, -22.371, 8.218, -148.169]
  MoveJ (Pt 12 (S136)) to (-437.91, 304.62, 83.06) mm, rotated rx 148.82 ry 3.26 rz -178.93 deg; joints [-75.565, -105.059, 145.828, -26.927, 13.754, -134.641]

--- program Pickupm5ToFaceTarget1 (robot UR10e) ---
  MoveJ (Pt 1 (S136)) to (-437.91, 304.62, 83.06) mm, rotated rx 148.82 ry 3.26 rz -178.93 deg; joints [-75.565, -105.059, 145.828, -26.927, 13.754, -134.641]
  MoveJ (Pt 2 (S195)) to (-424.05, 221.6, 32.68) mm, rotated rx 148.94 ry 3.77 rz -174.12 deg; joints [-76.807, -103.326, 153.048, -22.371, 8.218, -148.169]
  MoveJ (Pt 3 (S994)) to (-457.25, 218.7, 30) mm, rotated rx 148.82 ry 3.26 rz -178.93 deg; joints [-63.329, -105.109, 152.954, 319.665, 25.798, -127.95]
  MoveJ (Pt 4 (S1100)) to (-556.88, -13.22, 34.94) mm, rotated rx 135 ry 0 rz -90 deg; joints [-49.771, -80.79, 137.167, 303.621, -49.77, -134.999]
  MoveJ (Pt 5 (S1273)) to (-716.01, -98.69, 181.83) mm, rotated rx 90 ry 0 rz -90 deg; joints [-33.401, -75.109, 130.821, 304.286, -33.399, -179.998]
  MoveJ (Pt 6 (S1304)) to (-716.01, -59.98, 245.4) mm, rotated rx 90 ry 0 rz -90 deg; joints [-37.136, -80.295, 127.654, 312.639, -37.135, -179.998]
  MoveJ (Pt 7 (S1320)) to (-716.01, -159.98, 245.4) mm, rotated rx 90 ry 0 rz -90 deg; joints [-26.988, -82.105, 129.904, 312.198, -26.987, -179.998]
  MoveJ (Pt 8 (S1415)) to (-816.01, -159.98, 395.4) mm, rotated rx 90 ry 0 rz -90 deg; joints [-22.388, -83.255, 112.006, 331.246, -22.387, -179.997]
  MoveJ (Pt 9 (S1557)) to (-816.01, -159.98, 645.4) mm, rotated rx 90 ry 0 rz -90 deg; joints [-22.388, -89.789, 92.704, 357.083, -22.387, -179.997]
  MoveJ (Pt 10 (S1426)) to (-839.72, -113.23, 459.2) mm, rotated rx 135 ry 0 rz -90 deg; joints [-23.236, -80.609, 85.748, 354.857, -23.235, -134.997]
  MoveJ (Pt 11 (S1377)) to (-910.43, -113.22, 388.49) mm, rotated rx 135 ry 0 rz -90 deg; joints [-21.07, -72.993, 83.411, 349.579, -21.069, -134.997]
  MoveJ (Pt 12 (S1390)) to (-910.43, -13.22, 388.49) mm, rotated rx 135 ry 0 rz -90 deg; joints [-28.011, -71.089, 80.867, 350.219, -28.01, -134.998]

--- program FaceTarget2ToPickupm5 (robot UR10e) ---
  MoveJ (Pt 1 (S1558)) to (-1103.52, -62.25, 481.99) mm, rotated rx 180 ry 0 rz 173.43 deg; joints [-5.588, -58.826, 71.227, 167.599, -90.985, -270.001]
  MoveJ (Pt 2 (S1535)) to (-1100.79, -83.02, 481.99) mm, rotated rx 180 ry 0 rz 180 deg; joints [-5.882, -59.281, 71.94, 167.342, -84.119, -270.001]
  MoveJ (Pt 3 (S1520)) to (-1086.49, -83.02, 481.99) mm, rotated rx 180 ry 0 rz 180 deg; joints [-5.98, -60.665, 74.085, 166.58, -84.021, -270.001]
  MoveJ (Pt 4 (S1500)) to (-1087.69, 17.1, 481.99) mm, rotated rx -180 ry 0 rz 180 deg; joints [-12.597, -60.926, 74.486, 166.439, -77.405, -270]
  MoveJ (Pt 5 (S1429)) to (-587.69, -82.91, 481.99) mm, rotated rx -180 ry 0 rz 180 deg; joints [-14.522, -109.656, 127.541, 162.115, -75.48, -270]
  MoveJ (Pt 6 (S1089)) to (-587.69, -82.9, -18.01) mm, rotated rx -180 ry 0 rz 180 deg; joints [-14.523, -50.121, 145.657, 84.464, -75.479, -270]
  MoveJ (Pt 7 (S204)) to (-437.41, 306.44, 84.14) mm, rotated rx 148.94 ry 3.76 rz -174.12 deg; joints [-78.226, -98.327, 142.765, -11.769, 6.987, -153.532]
  MoveJ (Pt 8 (S195)) to (-424.05, 221.6, 32.68) mm, rotated rx 148.94 ry 3.77 rz -174.12 deg; joints [-76.807, -103.326, 153.048, -22.371, 8.218, -148.169]
  MoveJ (Pt 9 (S136)) to (-437.91, 304.62, 83.06) mm, rotated rx 148.82 ry 3.26 rz -178.93 deg; joints [-75.565, -105.059, 145.828, -26.927, 13.754, -134.641]

--- program Pickupm5ToFaceTarget2 (robot UR10e) ---
  MoveJ (Pt 1 (S136)) to (-437.91, 304.62, 83.06) mm, rotated rx 148.82 ry 3.26 rz -178.93 deg; joints [-75.565, -105.059, 145.828, -26.927, 13.754, -134.641]
  MoveJ (Pt 2 (S195)) to (-424.05, 221.6, 32.68) mm, rotated rx 148.94 ry 3.77 rz -174.12 deg; joints [-76.807, -103.326, 153.048, -22.371, 8.218, -148.169]
  MoveJ (Pt 3 (S204)) to (-437.41, 306.44, 84.14) mm, rotated rx 148.94 ry 3.76 rz -174.12 deg; joints [-78.226, -98.327, 142.765, -11.769, 6.987, -153.532]
  MoveJ (Pt 4 (S1089)) to (-587.69, -82.9, -18.01) mm, rotated rx -180 ry 0 rz 180 deg; joints [-14.523, -50.121, 145.657, 84.464, -75.479, -270]
  MoveJ (Pt 5 (S1429)) to (-587.69, -82.91, 481.99) mm, rotated rx -180 ry 0 rz 180 deg; joints [-14.522, -109.656, 127.541, 162.115, -75.48, -270]
  MoveJ (Pt 6 (S1522)) to (-1087.69, -82.9, 481.99) mm, rotated rx -180 ry 0 rz 180 deg; joints [-5.98, -60.551, 73.909, 166.641, -84.022, -270]
  MoveJ (Pt 7 (S1535)) to (-1100.79, -83.02, 481.99) mm, rotated rx 180 ry 0 rz 180 deg; joints [-5.882, -59.281, 71.94, 167.342, -84.119, -270.001]
  MoveJ (Pt 8 (S1558)) to (-1103.52, -62.25, 481.99) mm, rotated rx 180 ry 0 rz 173.43 deg; joints [-5.588, -58.826, 71.227, 167.599, -90.985, -270.001]

--- program Program_Face_0_m5 (robot UR10e) ---
  Call screw_in(0)
  Call Pickupm8ToFaceTarget0
  MoveL (Face_Target_0)
  MoveL (H-5.2_15.0-0)
  MoveL (Face_Target_0)
  Call FaceTarget0ToPickupm8

--- program Program_Face_1_m5 (robot UR10e) ---
  Call screw_in(0)
  Call Pickupm5ToFaceTarget1
  MoveL (Face_Target_1)
  MoveL (H-5.2_15.0-10)
  Call screw_in(20)
  Call screw_out(0)
  MoveL (Face_Target_1)
  Call FaceTarget1ToPickupm5
  Call screw_in(0)
  Call Pickupm5ToFaceTarget1
  MoveL (Face_Target_1)
  MoveL (H-5.2_15.0-11)
  Call screw_in(20)
  Call screw_out(0)
  MoveL (Face_Target_1)
  Call FaceTarget1ToPickupm5
  Call screw_in(0)
  Call Pickupm5ToFaceTarget1
  MoveL (Face_Target_1)
  MoveL (H-5.2_15.0-12)
  Call screw_in(20)
  Call screw_out(0)
  MoveL (Face_Target_1)
  Call FaceTarget1ToPickupm5
  Call screw_in(0)
  Call Pickupm5ToFaceTarget1
  MoveL (Face_Target_1)
  MoveL (H-5.2_15.0-15)
  Call screw_in(20)
  Call screw_out(0)
  MoveL (Face_Target_1)
  Call FaceTarget1ToPickupm5
  Call screw_in(0)

--- program Program_Face_2_m5 (robot UR10e) ---
  Call screw_in(0)
  Call Pickupm5ToFaceTarget2
  MoveL (Face_Target_2)
  MoveL (H-5.2_15.0-16)
  Call screw_in(20)
  Call screw_out(0)
  MoveL (Face_Target_2)
  Call FaceTarget2ToPickupm5
  Call screw_in(0)
  Call Pickupm5ToFaceTarget2
  MoveL (Face_Target_2)
  MoveL (H-5.2_15.0-17)
  Call screw_in(20)
  Call screw_out(0)
  MoveL (Face_Target_2)
  Call FaceTarget2ToPickupm5
  Call screw_in(0)
  Call Pickupm5ToFaceTarget2
  MoveL (Face_Target_2)
  MoveL (H-5.2_15.0-19)
  Call screw_in(20)
  Call screw_out(0)
  MoveL (Face_Target_2)
  Call FaceTarget2ToPickupm5
  Call screw_in(0)

--- program Program_Main_m8 (robot UR10e) ---
  Set Tool: schroevendraaier all in met nieuw kopstuk en tool
  Set Ref.: CSV Frame
  Call Program_Face_0_m8
  Call Program_Face_1_m8
  Call Program_Face_2_m8

--- program Program_Main_m5 (robot UR10e) ---
  Set Tool: schroevendraaier all in met nieuw kopstuk en tool
  Set Ref.: CSV Frame
  Call Program_Face_0_m5
  Call Program_Face_1_m5
  Call Program_Face_2_m5

--- program pickupm8Totoolswitchm8approach (robot UR10e) ---
  MoveJ (Pt 1 (S1245)) to (-361.97, 306.04, 87.38) mm, rotated rx 148.82 ry 3.26 rz -178.93 deg; joints [-96.274, -127.938, 155.828, 308.074, -8.028, -97.355]
  MoveJ (Pt 2 (S1259)) to (-291.81, 189.68, 43.36) mm, rotated rx 173.25 ry 30.68 rz -107.38 deg; joints [-75.824, -114.001, 145.678, 293.478, -63.249, -79.354]
  MoveJ (Pt 3 (S1095)) to (-362.69, 295.7, 104.49) mm, rotated rx 173.25 ry 30.68 rz -107.38 deg; joints [-70.201, -101.671, 131.181, 293.82, -58.685, -75.597]
  MoveJ (Pt 4 (S1043)) to (-433.56, 401.71, 165.63) mm, rotated rx 173.25 ry 30.68 rz -107.38 deg; joints [-67.129, -91.484, 115.69, 297.937, -56.239, -73.391]
  MoveJ (Pt 5 (S1113)) to (-437.47, 349.85, 251.04) mm, rotated rx 173.25 ry 30.68 rz -107.38 deg; joints [-64.592, -98.205, 112.824, 306.43, -54.251, -71.473]
  MoveJ (Pt 6 (S1127)) to (-539.86, 560.74, 257.33) mm, rotated rx 173.25 ry 30.68 rz -107.38 deg; joints [-64.444, -76.48, 89.354, 308.108, -54.136, -71.358]
  MoveJ (Pt 7 (S1511)) to (-816, 401.32, 181.84) mm, rotated rx 90 ry 0 rz -90 deg; joints [-57.758, -50.359, 88.357, 322, -57.757, -179.999]
  MoveJ (Pt 8 (S1345)) to (-816, 151.32, 181.83) mm, rotated rx 90 ry 0 rz -90 deg; joints [-46.116, -61.68, 108.893, 312.786, -46.115, -179.999]
  MoveJ (Pt 9 (S1313)) to (-816, 90.03, 145.4) mm, rotated rx 90 ry 0 rz -90 deg; joints [-42.32, -60.916, 113.175, 307.739, -42.319, -179.999]
  MoveJ (Pt 10 (S901)) to (-623.37, -125.97, 47.51) mm, rotated rx -179.93 ry 0 rz -89.98 deg; joints [-24.394, -73.129, 114.763, 318.368, -24.416, -89.927]
  MoveJ (Pt 11 (S928)) to (-624.14, -217.54, 76.08) mm, rotated rx -179.87 ry 0.01 rz -89.96 deg; joints [-16.172, -75.486, 114.259, 321.203, -16.217, -89.845]
  MoveJ (Pt 12 (S933)) to (-624.02, -367.54, 76.06) mm, rotated rx -179.87 ry 0.01 rz -89.96 deg; joints [-2.191, -74.037, 112.291, 321.575, -2.235, -89.697]
  MoveJ (Pt 13 (S978)) to (-723.79, -367.61, -24.17) mm, rotated rx -179.87 ry 0.01 rz -89.96 deg; joints [-1.881, -60.061, 103.916, 315.946, -1.925, -89.669]
  MoveJ (Pt 14 (S1025)) to (-723.71, -467.61, -24.18) mm, rotated rx -179.87 ry 0.01 rz -89.96 deg; joints [5.95, -58.113, 100.501, 317.677, 5.906, -89.932]
  MoveJ (Pt 15 (S1056)) to (-723.94, -467.62, 75.82) mm, rotated rx -179.87 ry 0.01 rz -89.96 deg; joints [5.949, -63.92, 97.407, 326.578, 5.905, -89.932]
  MoveJ (Pt 16 (S940)) to (-623.94, -467.54, 76.05) mm, rotated rx -179.87 ry 0.01 rz -89.96 deg; joints [6.859, -71.505, 108.744, 322.817, 6.815, -89.924]

--- program toolswitchm8approachTopickupm8 (robot UR10e) ---
  MoveJ (Pt 1 (S940)) to (-623.94, -467.54, 76.05) mm, rotated rx -179.87 ry 0.01 rz -89.96 deg; joints [6.859, -71.505, 108.744, 322.817, 6.815, -89.924]
  MoveJ (Pt 2 (S1056)) to (-723.94, -467.62, 75.82) mm, rotated rx -179.87 ry 0.01 rz -89.96 deg; joints [5.949, -63.92, 97.407, 326.578, 5.905, -89.932]
  MoveJ (Pt 3 (S1025)) to (-723.71, -467.61, -24.18) mm, rotated rx -179.87 ry 0.01 rz -89.96 deg; joints [5.95, -58.113, 100.501, 317.677, 5.906, -89.932]
  MoveJ (Pt 4 (S978)) to (-723.79, -367.61, -24.17) mm, rotated rx -179.87 ry 0.01 rz -89.96 deg; joints [-1.881, -60.061, 103.916, 315.946, -1.925, -89.669]
  MoveJ (Pt 5 (S933)) to (-624.02, -367.54, 76.06) mm, rotated rx -179.87 ry 0.01 rz -89.96 deg; joints [-2.191, -74.037, 112.291, 321.575, -2.235, -89.697]
  MoveJ (Pt 6 (S928)) to (-624.14, -217.54, 76.08) mm, rotated rx -179.87 ry 0.01 rz -89.96 deg; joints [-16.172, -75.486, 114.259, 321.203, -16.217, -89.845]
  MoveJ (Pt 7 (S901)) to (-623.37, -125.97, 47.51) mm, rotated rx -179.93 ry 0 rz -89.98 deg; joints [-24.394, -73.129, 114.763, 318.368, -24.416, -89.927]
  MoveJ (Pt 8 (S1313)) to (-816, 90.03, 145.4) mm, rotated rx 90 ry 0 rz -90 deg; joints [-42.32, -60.916, 113.175, 307.739, -42.319, -179.999]
  MoveJ (Pt 9 (S1345)) to (-816, 151.32, 181.83) mm, rotated rx 90 ry 0 rz -90 deg; joints [-46.116, -61.68, 108.893, 312.786, -46.115, -179.999]
  MoveJ (Pt 10 (S1511)) to (-816, 401.32, 181.84) mm, rotated rx 90 ry 0 rz -90 deg; joints [-57.758, -50.359, 88.357, 322, -57.757, -179.999]
  MoveJ (Pt 11 (S1127)) to (-539.86, 560.74, 257.33) mm, rotated rx 173.25 ry 30.68 rz -107.38 deg; joints [-64.444, -76.48, 89.354, 308.108, -54.136, -71.358]
  MoveJ (Pt 12 (S1113)) to (-437.47, 349.85, 251.04) mm, rotated rx 173.25 ry 30.68 rz -107.38 deg; joints [-64.592, -98.205, 112.824, 306.43, -54.251, -71.473]
  MoveJ (Pt 13 (S1043)) to (-433.56, 401.71, 165.63) mm, rotated rx 173.25 ry 30.68 rz -107.38 deg; joints [-67.129, -91.484, 115.69, 297.937, -56.239, -73.391]
  MoveJ (Pt 14 (S1095)) to (-362.69, 295.7, 104.49) mm, rotated rx 173.25 ry 30.68 rz -107.38 deg; joints [-70.201, -101.671, 131.181, 293.82, -58.685, -75.597]
  MoveJ (Pt 15 (S1259)) to (-291.81, 189.68, 43.36) mm, rotated rx 173.25 ry 30.68 rz -107.38 deg; joints [-75.824, -114.001, 145.678, 293.478, -63.249, -79.354]
  MoveJ (Pt 16 (S1245)) to (-361.97, 306.04, 87.38) mm, rotated rx 148.82 ry 3.26 rz -178.93 deg; joints [-96.274, -127.938, 155.828, 308.074, -8.028, -97.355]

--- program Tool_Pickup_m8 (robot UR10e) ---
  Call pickupm8Totoolswitchm8approach
  MoveL (toolswitch_m8)
  Call screw_out(0)
  MoveL (toolswitch_m8_approach)
  Call toolswitchm8approachTopickupm8

--- program Tool_Dropoff_m8 (robot UR10e) ---
  Call pickupm8Totoolswitchm8approach
  MoveL (toolswitch_m8)
  Call screw_in(10)
  MoveL (toolswitch_m8_approach)
  Call toolswitchm8approachTopickupm8

--- program pickupm5Totoolswitchm5approach (robot UR10e) ---
  MoveJ (Pt 1 (S136)) to (-437.91, 304.62, 83.06) mm, rotated rx 148.82 ry 3.26 rz -178.93 deg; joints [-75.565, -105.059, 145.828, -26.927, 13.754, -134.641]
  MoveJ (Pt 2 (S195)) to (-424.05, 221.6, 32.68) mm, rotated rx 148.94 ry 3.77 rz -174.12 deg; joints [-76.807, -103.326, 153.048, -22.371, 8.218, -148.169]
  MoveJ (Pt 3 (S994)) to (-457.25, 218.7, 30) mm, rotated rx 148.82 ry 3.26 rz -178.93 deg; joints [-63.329, -105.109, 152.954, 319.665, 25.798, -127.95]
  MoveJ (Pt 4 (S1100)) to (-556.88, -13.22, 34.94) mm, rotated rx 135 ry 0 rz -90 deg; joints [-49.771, -80.79, 137.167, 303.621, -49.77, -134.999]
  MoveJ (Pt 5 (S1370)) to (-556.88, -13.23, 388.49) mm, rotated rx 135 ry 0 rz -90 deg; joints [-49.771, -103.763, 115.12, 348.641, -49.77, -134.999]
  MoveJ (Pt 6 (S1170)) to (-373.69, -125.87, 297.83) mm, rotated rx -179.93 ry 0 rz -89.98 deg; joints [-40.714, -110.761, 122.459, 348.303, -40.737, -89.926]
  MoveJ (Pt 7 (S1200)) to (-374.71, -217.38, 326.65) mm, rotated rx -179.87 ry 0.01 rz -89.96 deg; joints [-27.681, -112.486, 120.555, 351.916, -27.726, -89.855]
  MoveJ (Pt 8 (S1384)) to (-556.88, -263.23, 388.48) mm, rotated rx 135 ry 0 rz -90 deg; joints [-19.023, -108.994, 118.744, 350.247, -19.022, -134.996]
  MoveJ (Pt 9 (S1171)) to (-733.66, -263.22, 211.71) mm, rotated rx 135 ry 0 rz -90 deg; joints [-12.934, -83.618, 115.657, 327.956, -12.933, -134.995]
  MoveJ (Pt 10 (S928)) to (-624.14, -217.54, 76.08) mm, rotated rx -179.87 ry 0.01 rz -89.96 deg; joints [-16.172, -75.486, 114.259, 321.203, -16.217, -89.845]
  MoveJ (Pt 11 (S933)) to (-624.02, -367.54, 76.06) mm, rotated rx -179.87 ry 0.01 rz -89.96 deg; joints [-2.191, -74.037, 112.291, 321.575, -2.235, -89.697]
  MoveJ (Pt 12 (S903)) to (-623.27, -375.97, 47.51) mm, rotated rx -179.93 ry 0 rz -89.98 deg; joints [-1.416, -72.071, 113.252, 318.849, -1.438, -89.956]

--- program toolswitchm5approachTopickupm5 (robot UR10e) ---
  MoveJ (Pt 1 (S903)) to (-623.27, -375.97, 47.51) mm, rotated rx -179.93 ry 0 rz -89.98 deg; joints [-1.416, -72.071, 113.252, 318.849, -1.438, -89.956]
  MoveJ (Pt 2 (S933)) to (-624.02, -367.54, 76.06) mm, rotated rx -179.87 ry 0.01 rz -89.96 deg; joints [-2.191, -74.037, 112.291, 321.575, -2.235, -89.697]
  MoveJ (Pt 3 (S928)) to (-624.14, -217.54, 76.08) mm, rotated rx -179.87 ry 0.01 rz -89.96 deg; joints [-16.172, -75.486, 114.259, 321.203, -16.217, -89.845]
  MoveJ (Pt 4 (S1171)) to (-733.66, -263.22, 211.71) mm, rotated rx 135 ry 0 rz -90 deg; joints [-12.934, -83.618, 115.657, 327.956, -12.933, -134.995]
  MoveJ (Pt 5 (S1384)) to (-556.88, -263.23, 388.48) mm, rotated rx 135 ry 0 rz -90 deg; joints [-19.023, -108.994, 118.744, 350.247, -19.022, -134.996]
  MoveJ (Pt 6 (S1200)) to (-374.71, -217.38, 326.65) mm, rotated rx -179.87 ry 0.01 rz -89.96 deg; joints [-27.681, -112.486, 120.555, 351.916, -27.726, -89.855]
  MoveJ (Pt 7 (S1170)) to (-373.69, -125.87, 297.83) mm, rotated rx -179.93 ry 0 rz -89.98 deg; joints [-40.714, -110.761, 122.459, 348.303, -40.737, -89.926]
  MoveJ (Pt 8 (S1370)) to (-556.88, -13.23, 388.49) mm, rotated rx 135 ry 0 rz -90 deg; joints [-49.771, -103.763, 115.12, 348.641, -49.77, -134.999]
  MoveJ (Pt 9 (S1100)) to (-556.88, -13.22, 34.94) mm, rotated rx 135 ry 0 rz -90 deg; joints [-49.771, -80.79, 137.167, 303.621, -49.77, -134.999]
  MoveJ (Pt 10 (S994)) to (-457.25, 218.7, 30) mm, rotated rx 148.82 ry 3.26 rz -178.93 deg; joints [-63.329, -105.109, 152.954, 319.665, 25.798, -127.95]
  MoveJ (Pt 11 (S195)) to (-424.05, 221.6, 32.68) mm, rotated rx 148.94 ry 3.77 rz -174.12 deg; joints [-76.807, -103.326, 153.048, -22.371, 8.218, -148.169]
  MoveJ (Pt 12 (S136)) to (-437.91, 304.62, 83.06) mm, rotated rx 148.82 ry 3.26 rz -178.93 deg; joints [-75.565, -105.059, 145.828, -26.927, 13.754, -134.641]

--- program Tool_Pickup_m5 (robot UR10e) ---
  Call pickupm8Totoolswitchm5approach
  MoveL (toolswitch_m5_approach)
  MoveL (toolswitch_m5)
  Call screw_out(0)
  MoveL (toolswitch_m5_approach)
  Call toolswitchm5approachTopickupm8

--- program Tool_Dropoff_m5 (robot UR10e) ---
  Call pickupm8Totoolswitchm5approach
  MoveL (toolswitch_m5)
  Call screw_in(10)
  MoveL (toolswitch_m5_approach)
  Call toolswitchm5approachTopickupm8

--- program Program_Main_Combined (robot UR10e) ---
  Set Tool: schroevendraaier all in met nieuw kopstuk en tool
  Set Ref.: CSV Frame
  Call Tool_Pickup_m8
  Call Program_Main_m8
  Call Tool_Dropoff_m8
  Call Tool_Pickup_m5
  Call Program_Face_0_m5
  Call Tool_Dropoff_m5

--- program toolswitchm5approachTopickupm8 (robot UR10e) ---
  MoveJ (Pt 1 (S903)) to (-623.27, -375.97, 47.51) mm, rotated rx -179.93 ry 0 rz -89.98 deg; joints [-1.416, -72.071, 113.252, 318.849, -1.438, -89.956]
  MoveJ (Pt 2 (S933)) to (-624.02, -367.54, 76.06) mm, rotated rx -179.87 ry 0.01 rz -89.96 deg; joints [-2.191, -74.037, 112.291, 321.575, -2.235, -89.697]
  MoveJ (Pt 3 (S928)) to (-624.14, -217.54, 76.08) mm, rotated rx -179.87 ry 0.01 rz -89.96 deg; joints [-16.172, -75.486, 114.259, 321.203, -16.217, -89.845]
  MoveJ (Pt 4 (S901)) to (-623.37, -125.97, 47.51) mm, rotated rx -179.93 ry 0 rz -89.98 deg; joints [-24.394, -73.129, 114.763, 318.368, -24.416, -89.927]
  MoveJ (Pt 5 (S1313)) to (-816, 90.03, 145.4) mm, rotated rx 90 ry 0 rz -90 deg; joints [-42.32, -60.916, 113.175, 307.739, -42.319, -179.999]
  MoveJ (Pt 6 (S1345)) to (-816, 151.32, 181.83) mm, rotated rx 90 ry 0 rz -90 deg; joints [-46.116, -61.68, 108.893, 312.786, -46.115, -179.999]
  MoveJ (Pt 7 (S1511)) to (-816, 401.32, 181.84) mm, rotated rx 90 ry 0 rz -90 deg; joints [-57.758, -50.359, 88.357, 322, -57.757, -179.999]
  MoveJ (Pt 8 (S1127)) to (-539.86, 560.74, 257.33) mm, rotated rx 173.25 ry 30.68 rz -107.38 deg; joints [-64.444, -76.48, 89.354, 308.108, -54.136, -71.358]
  MoveJ (Pt 9 (S1113)) to (-437.47, 349.85, 251.04) mm, rotated rx 173.25 ry 30.68 rz -107.38 deg; joints [-64.592, -98.205, 112.824, 306.43, -54.251, -71.473]
  MoveJ (Pt 10 (S1043)) to (-433.56, 401.71, 165.63) mm, rotated rx 173.25 ry 30.68 rz -107.38 deg; joints [-67.129, -91.484, 115.69, 297.937, -56.239, -73.391]
  MoveJ (Pt 11 (S1095)) to (-362.69, 295.7, 104.49) mm, rotated rx 173.25 ry 30.68 rz -107.38 deg; joints [-70.201, -101.671, 131.181, 293.82, -58.685, -75.597]
  MoveJ (Pt 12 (S1259)) to (-291.81, 189.68, 43.36) mm, rotated rx 173.25 ry 30.68 rz -107.38 deg; joints [-75.824, -114.001, 145.678, 293.478, -63.249, -79.354]
  MoveJ (Pt 13 (S1245)) to (-361.97, 306.04, 87.38) mm, rotated rx 148.82 ry 3.26 rz -178.93 deg; joints [-96.274, -127.938, 155.828, 308.074, -8.028, -97.355]

--- program pickupm8Totoolswitchm5approach (robot UR10e) ---
  MoveJ (Pt 1 (S1245)) to (-361.97, 306.04, 87.38) mm, rotated rx 148.82 ry 3.26 rz -178.93 deg; joints [-96.274, -127.938, 155.828, 308.074, -8.028, -97.355]
  MoveJ (Pt 2 (S1259)) to (-291.81, 189.68, 43.36) mm, rotated rx 173.25 ry 30.68 rz -107.38 deg; joints [-75.824, -114.001, 145.678, 293.478, -63.249, -79.354]
  MoveJ (Pt 3 (S1095)) to (-362.69, 295.7, 104.49) mm, rotated rx 173.25 ry 30.68 rz -107.38 deg; joints [-70.201, -101.671, 131.181, 293.82, -58.685, -75.597]
  MoveJ (Pt 4 (S1043)) to (-433.56, 401.71, 165.63) mm, rotated rx 173.25 ry 30.68 rz -107.38 deg; joints [-67.129, -91.484, 115.69, 297.937, -56.239, -73.391]
  MoveJ (Pt 5 (S1113)) to (-437.47, 349.85, 251.04) mm, rotated rx 173.25 ry 30.68 rz -107.38 deg; joints [-64.592, -98.205, 112.824, 306.43, -54.251, -71.473]
  MoveJ (Pt 6 (S1127)) to (-539.86, 560.74, 257.33) mm, rotated rx 173.25 ry 30.68 rz -107.38 deg; joints [-64.444, -76.48, 89.354, 308.108, -54.136, -71.358]
  MoveJ (Pt 7 (S1511)) to (-816, 401.32, 181.84) mm, rotated rx 90 ry 0 rz -90 deg; joints [-57.758, -50.359, 88.357, 322, -57.757, -179.999]
  MoveJ (Pt 8 (S1345)) to (-816, 151.32, 181.83) mm, rotated rx 90 ry 0 rz -90 deg; joints [-46.116, -61.68, 108.893, 312.786, -46.115, -179.999]
  MoveJ (Pt 9 (S1313)) to (-816, 90.03, 145.4) mm, rotated rx 90 ry 0 rz -90 deg; joints [-42.32, -60.916, 113.175, 307.739, -42.319, -179.999]
  MoveJ (Pt 10 (S901)) to (-623.37, -125.97, 47.51) mm, rotated rx -179.93 ry 0 rz -89.98 deg; joints [-24.394, -73.129, 114.763, 318.368, -24.416, -89.927]
  MoveJ (Pt 11 (S928)) to (-624.14, -217.54, 76.08) mm, rotated rx -179.87 ry 0.01 rz -89.96 deg; joints [-16.172, -75.486, 114.259, 321.203, -16.217, -89.845]
  MoveJ (Pt 12 (S933)) to (-624.02, -367.54, 76.06) mm, rotated rx -179.87 ry 0.01 rz -89.96 deg; joints [-2.191, -74.037, 112.291, 321.575, -2.235, -89.697]
  MoveJ (Pt 13 (S903)) to (-623.27, -375.97, 47.51) mm, rotated rx -179.93 ry 0 rz -89.98 deg; joints [-1.416, -72.071, 113.252, 318.849, -1.438, -89.956]
